FUNCTION_BLOCK SimpleButtonWithHold
VAR_INPUT
END_VAR
VAR_OUTPUT
END_VAR
VAR
END_VAR

END_FUNCTION_BLOCK

(* stored: Version 1.1.0.1, ProductVersion 3.1.4024.12
   POU SimpleButtonWithHold: Id {f088760e-ef23-410b-b173-1afa982e1c6d}, SpecialFunc None *)
